{attribute 'GeneratedUsingTerminal: EJ5002-0000-0017'}
{attribute addProperty BoxType "EJ5002-0000-0017"}
{attribute addProperty Description "EJ5002 2Ch. SSI Encoder"}
{attribute addProperty Physics "KK"}
{attribute addProperty Id "SSI_Inputs_Channel_1AT %I*SSI_Inputs_Channel_EDA1628411SSI_Inputs_Channel_2AT %I*SSI_Inputs_Channel_EDA1628411WcStateAT %I*WcState_9091E0EB2InfoDataAT %I*InfoData_32EB74EA10"}
{attribute addProperty CRC "832804578"}
{attribute addProperty Size "34"}
TYPE EJ5002_31A396E2 EXTENDS EtcSlaveTerminalBase_947E5A46 :
STRUCT
	{attribute addProperty Name "SSI_Inputs_Channel_1"}
	SSI_Inputs_Channel_1 : SSI_Inputs_Channel_EDA16284;
	{attribute addProperty Name "SSI_Inputs_Channel_2"}
	SSI_Inputs_Channel_2 : SSI_Inputs_Channel_EDA16284;
	{attribute addProperty Name "WcState"}
	WcState : WcState_9091E0EB;
	{attribute addProperty Name "InfoData"}
	InfoData : InfoData_32EB74EA;
END_STRUCT
END_TYPE

(* stored: Version 1.2.0.0, ProductVersion 3.1.4024.9
   DUT EJ5002_31A396E2: Id {6ec28b49-2b0a-4f2f-9725-25da2f0d3d48} *)
